TYPE ST_HartingIO_get :
STRUCT
	b_DigitalInput1Active		:	BOOL;
	b_DigitalInput2Active		:	BOOL;
	b_GenLowFuel				:	BOOL;
	b_ExtSystemShutdownRequest	:	BOOL;
	b_ExtEMstopOK				: 	BOOL;
	b_ExtEMstopActive			: 	BOOL;
END_STRUCT
END_TYPE

(* stored: Version 1.1.0.1, ProductVersion 3.1.4026.18
   DUT ST_HartingIO_get: Id {031a363a-69e2-4dee-992f-dda1bdce04ff} *)
